% RSLogix 500 project P7_BAK024.RSS, saved by version 8.10.00.18 %
PROJECT "UNTITLED"    % processor: Bul.1763 MicroLogix 1100 Series A %

PROGRAM FILES
  LAD 2   6 rungs
  LAD 3 "IO'S"  5 rungs
  LAD 4 "CONTROL"  3 rungs
  LAD 5 "CALIB"  8 rungs
  LAD 6 "CYCLE"  2 rungs

DATA FILES
  O0 OUTPUT  4 elements
  I1 INPUT  6 elements
  S2 STATUS  66 elements
  B3 BINARY  1 elements
  T4 TIMER  4 elements
  C5 COUNTER  2 elements
  R6 CONTROL  1 elements
  N7 INTEGER  8 elements
  F8 FLOAT  10 elements

LADDER 2
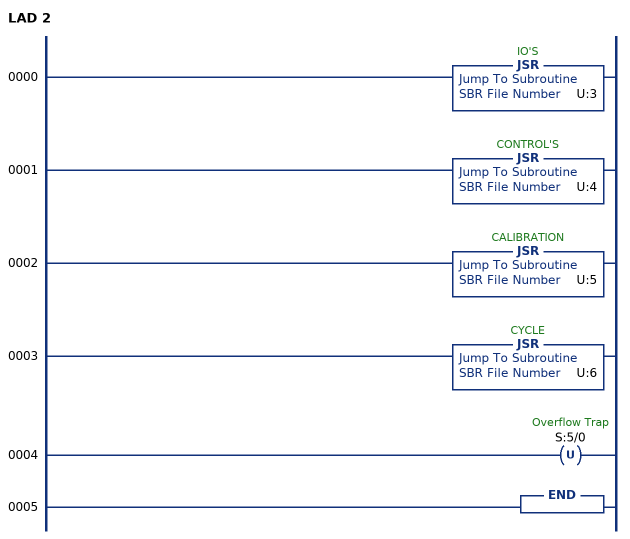
% Rung: 0 %
SOR JSR U:3 EOR
%   U:3  "IO'S" %
% Rung: 1 %
SOR JSR U:4 EOR
%   U:4  "CONTROL'S" %
% Rung: 2 %
SOR JSR U:5 EOR
%   U:5  "CALIBRATION" %
% Rung: 3 %
SOR JSR U:6 EOR
%   U:6  "CYCLE" %
% Rung: 4 %
SOR OTU S:5/0 EOR
%   S:5/0  "Overflow Trap" %
% Rung: 5 %
SOR END EOR

LADDER 3 "IO'S"
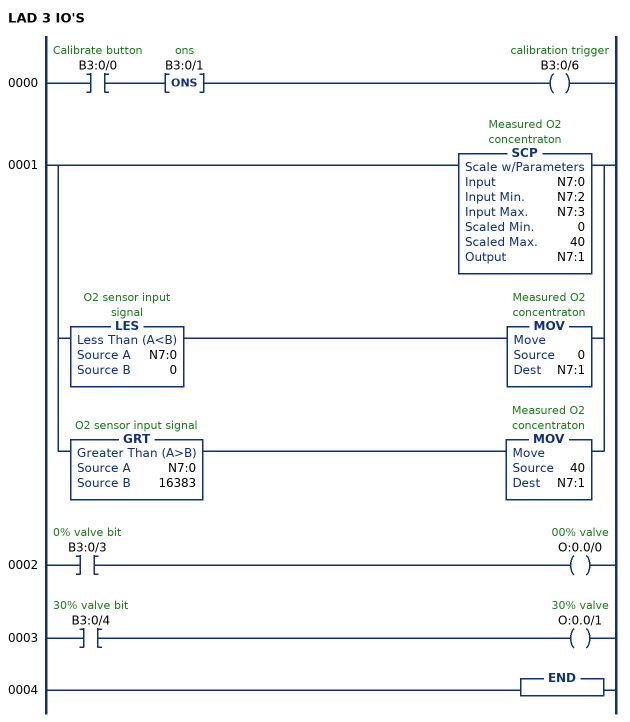
% Rung: 0 %
SOR XIC B3:0/0 ONS B3:0/1 OTE B3:0/6 EOR
%   B3:0/0  "Calibrate button" %
%   B3:0/1  "ons" %
%   B3:0/6  "calibration trigger" %
% Rung: 1 %
SOR BST SCP N7:0 N7:2 N7:3 0 40 N7:1 NXB LES N7:0 0 MOV 0 N7:1 NXB GRT N7:0 16383 MOV 40 N7:1 BND EOR
%   N7:0  "O2 sensor input signal" %
%   N7:2  "O2 input min" %
%   N7:3  "O2 input max" %
%   N7:1  "Measured O2 concentraton" %
% Rung: 2 %
SOR XIC B3:0/3 OTE O:0.0/0 EOR
%   B3:0/3  "0% valve bit" %
%   O:0.0/0  "00% valve" %
% Rung: 3 %
SOR XIC B3:0/4 OTE O:0.0/1 EOR
%   B3:0/4  "30% valve bit" %
%   O:0.0/1  "30% valve" %
% Rung: 4 %
SOR END EOR

LADDER 4 "CONTROL"
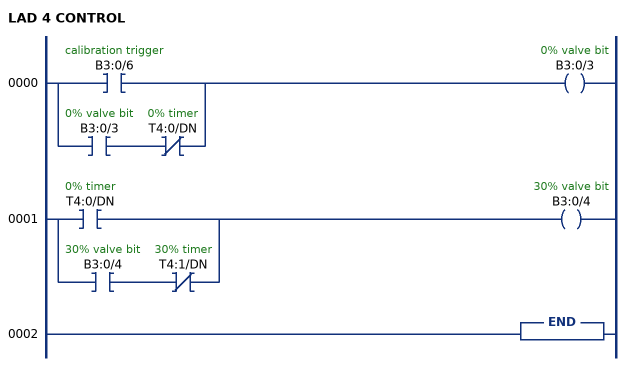
% Rung: 0 %
SOR BST XIC B3:0/6 NXB XIC B3:0/3 XIO T4:0/DN BND OTE B3:0/3 EOR
%   B3:0/6  "calibration trigger" %
%   B3:0/3  "0% valve bit" %
%   T4:0  "0% timer" %
% Rung: 1 %
SOR BST XIC T4:0/DN NXB XIC B3:0/4 XIO T4:1/DN BND OTE B3:0/4 EOR
%   T4:0  "0% timer" %
%   B3:0/4  "30% valve bit" %
%   T4:1  "30% timer" %
% Rung: 2 %
SOR END EOR

LADDER 5 "CALIB"
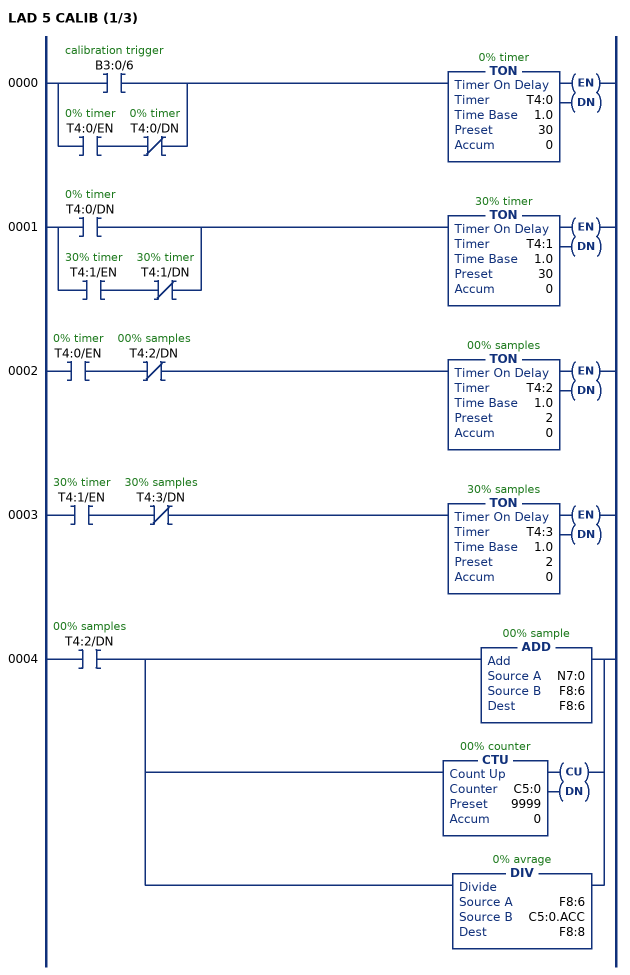
% Rung: 0 %
SOR BST XIC B3:0/6 NXB XIC T4:0/EN XIO T4:0/DN BND TON T4:0 1.0 30 0 EOR
%   B3:0/6  "calibration trigger" %
%   T4:0  "0% timer" %
% Rung: 1 %
SOR BST XIC T4:0/DN NXB XIC T4:1/EN XIO T4:1/DN BND TON T4:1 1.0 30 0 EOR
%   T4:0  "0% timer" %
%   T4:1  "30% timer" %
% Rung: 2 %
SOR XIC T4:0/EN XIO T4:2/DN TON T4:2 1.0 2 0 EOR
%   T4:0  "0% timer" %
%   T4:2  "00% samples" %
% Rung: 3 %
SOR XIC T4:1/EN XIO T4:3/DN TON T4:3 1.0 2 0 EOR
%   T4:1  "30% timer" %
%   T4:3  "30% samples" %
% Rung: 4 %
SOR XIC T4:2/DN BST ADD N7:0 F8:6 F8:6 NXB CTU C5:0 9999 0 NXB DIV F8:6 C5:0.ACC F8:8 BND EOR
%   T4:2  "00% samples" %
%   N7:0  "O2 sensor input signal" %
%   F8:6  "00% sample" %
%   C5:0  "00% counter" %
%   F8:8  "0% avrage" %

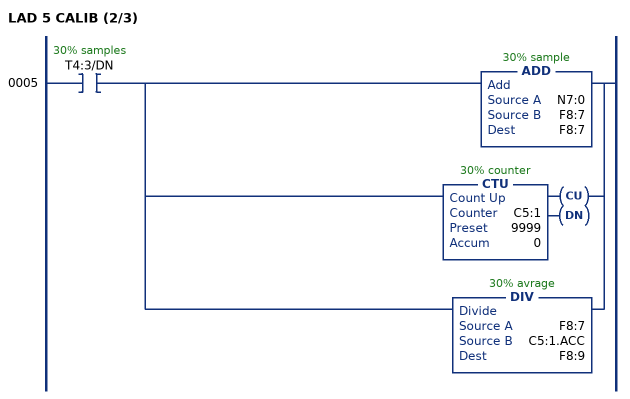
% Rung: 5 %
SOR XIC T4:3/DN BST ADD N7:0 F8:7 F8:7 NXB CTU C5:1 9999 0 NXB DIV F8:7 C5:1.ACC F8:9 BND EOR
%   T4:3  "30% samples" %
%   N7:0  "O2 sensor input signal" %
%   F8:7  "30% sample" %
%   C5:1  "30% counter" %
%   F8:9  "30% avrage" %

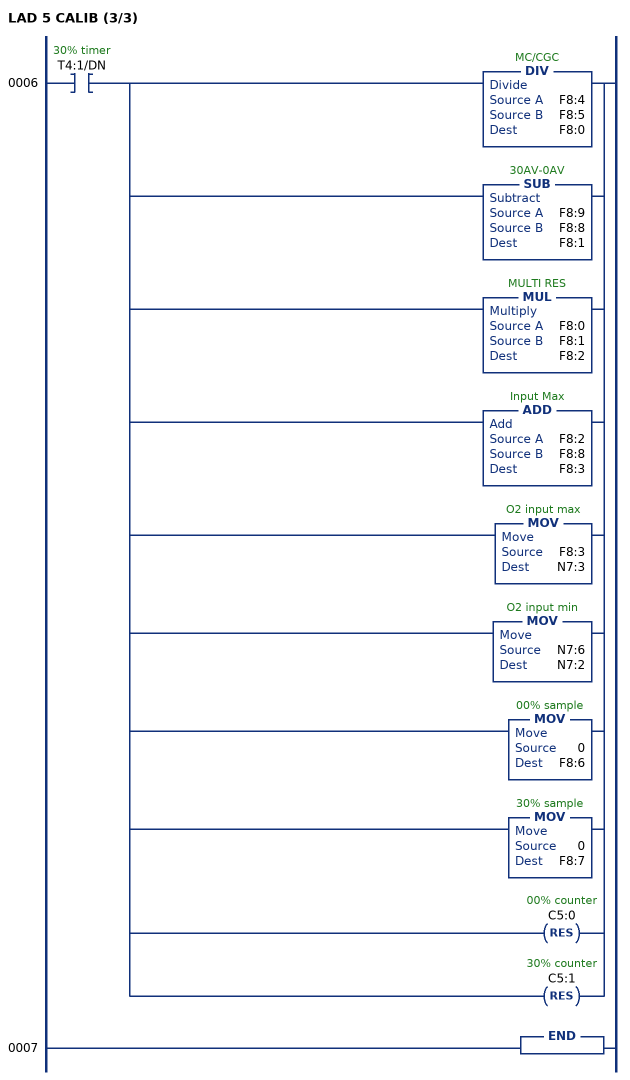
% Rung: 6 %
SOR XIC T4:1/DN BST DIV F8:4 F8:5 F8:0 NXB SUB F8:9 F8:8 F8:1 NXB MUL F8:0 F8:1 F8:2 NXB ADD F8:2 F8:8 F8:3 NXB MOV F8:3 N7:3 NXB MOV N7:6 N7:2 NXB MOV 0 F8:6 NXB MOV 0 F8:7 NXB RES C5:0 NXB RES C5:1 BND EOR
%   T4:1  "30% timer" %
%   F8:4  "40" %
%   F8:5  "30" %
%   F8:0  "MC/CGC" %
%   F8:9  "30% avrage" %
%   F8:8  "0% avrage" %
%   F8:1  "30AV-0AV" %
%   F8:2  "MULTI RES" %
%   F8:3  "Input Max" %
%   N7:3  "O2 input max" %
%   N7:6  "0% avrage" %
%   N7:2  "O2 input min" %
%   F8:6  "00% sample" %
%   F8:7  "30% sample" %
%   C5:0  "00% counter" %
%   C5:1  "30% counter" %
% Rung: 7 %
SOR END EOR

LADDER 6 "CYCLE"
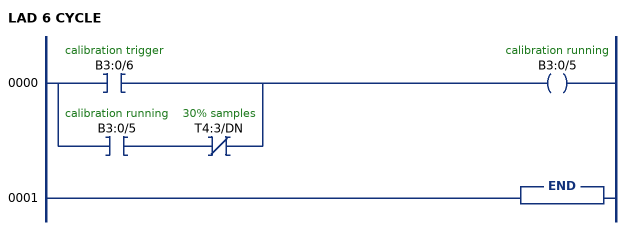
% Rung: 0 %
SOR BST XIC B3:0/6 NXB XIC B3:0/5 XIO T4:3/DN BND OTE B3:0/5 EOR
%   B3:0/6  "calibration trigger" %
%   B3:0/5  "calibration running" %
%   T4:3  "30% samples" %
% Rung: 1 %
SOR END EOR

OTHER DOCUMENTED ADDRESSES
  B3:0/2  "Calibrate Trigger"
  B3:0/7  "callibration interrupt"
  N7:4  "00% sampels"
  N7:5  "30% sample"
  N7:7  "30% avareg"

DATA TABLE (non-zero values as saved)
DATA T4
% .PRE .ACC %
% T4:0 % 30 0
% T4:1 % 30 0
% T4:2 % 2 0
% T4:3 % 2 0
DATA C5
% .PRE .ACC %
% C5:0 % 9999 0
% C5:1 % 9999 0
DATA N7
% N7:0 % 12288 0 0 0 0 0 0 0
DATA F8
% F8:0 % 1.333333 0 0 1092 40
% F8:5 % 30 0 0 12288 12288
